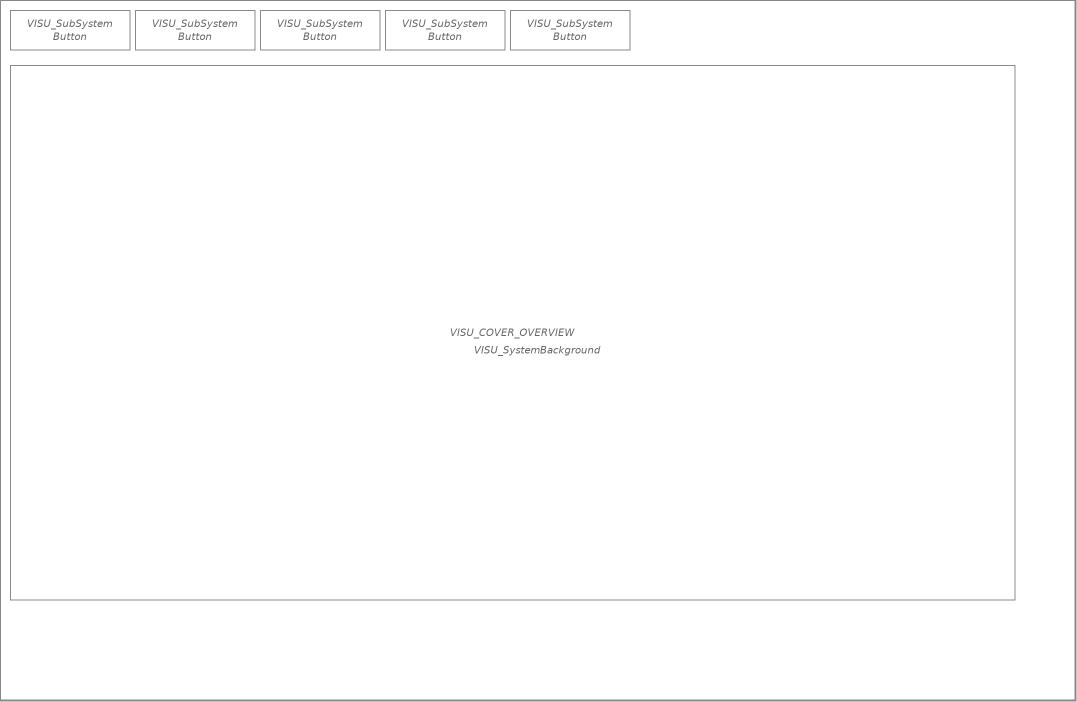
VISUALIZATION VISU_Cover  // 1077x702
VAR_IN_OUT
	ref : Cover;
    widget : CoverWidget;
END_VAR
    Frame (0,0 1075x700)
        shows VISU_SystemBackground(color := widget.actualStatus.color)
    Frame (10,65 1005x535)
        shows VISU_COVER_OVERVIEW(cover := ref, coverWidget := widget)
        shows VISU_CoverPanelSet(config := ref.config.top, set := ref.parts.top, widget := widget.top, currentMeasurement := ref.currentMeasurement)
        shows VISU_CoverPanelSet(config := ref.config.bottom, set := ref.parts.bottom, widget := widget.bottom, currentMeasurement := ref.currentMeasurement)
        shows VISU_CoverIO(io := ref.parts.io, widget := widget.io)
        shows VISU_CoverConfig(editableConfig := ref.editableConfig, activeConfig := ref.config, mgr := ref.parts.configManager, mgrWidget := widget.configManager, activeTab := widget.activeConfigTab)
    Frame (10,10 120x40)
        shows VISU_SubSystemButton(widget := widget.button_overview)
        OnMouseClick: FrameSelectionChange Selection=SelectedFrame=804c056d-b005-490b-b68c-1832c22506a3, GlobSel=AssignType=Directly, SelType=Locally
        OnMouseClick: execute { widget.activeTab := CoverTabs.OVERVIEW; }
    Frame (135,10 120x40)
        shows VISU_SubSystemButton(widget := widget.button_top)
        OnMouseClick: FrameSelectionChange Selection=SelectedFrame=804c056d-b005-490b-b68c-1832c22506a3, Selection=1, GlobSel=AssignType=Directly, SelType=Locally
        OnMouseClick: execute { widget.activeTab := CoverTabs.TOP; }
    Frame (260,10 120x40)
        shows VISU_SubSystemButton(widget := widget.button_bottom)
        OnMouseClick: FrameSelectionChange Selection=SelectedFrame=804c056d-b005-490b-b68c-1832c22506a3, Selection=2, GlobSel=AssignType=Directly, SelType=Locally
        OnMouseClick: execute { widget.activeTab := CoverTabs.BOTTOM; }
    Frame (385,10 120x40)
        shows VISU_SubSystemButton(widget := widget.button_io)
        OnMouseClick: FrameSelectionChange Selection=SelectedFrame=804c056d-b005-490b-b68c-1832c22506a3, Selection=3, GlobSel=AssignType=Directly, SelType=Locally
        OnMouseClick: execute { widget.activeTab := CoverTabs.IO; }
    Frame (510,10 120x40)
        shows VISU_SubSystemButton(widget := widget.button_config)
        OnMouseClick: FrameSelectionChange Selection=SelectedFrame=804c056d-b005-490b-b68c-1832c22506a3, Selection=4, GlobSel=AssignType=Directly, SelType=Locally
        OnMouseClick: execute { widget.activeTab := CoverTabs.CONFIG; }
END_VISUALIZATION

(* stored: Version 1.1.0.1, ProductVersion 3.1.4019.2
   Visu VISU_Cover: Id {e44c03c4-b5af-429b-a207-99f0b9b35bc5} *)
